// TIA Portal V20 export
// export: Created 2025-12-01T14:57:43.1405238Z, ExportSetting None, DisplayName Totally Integrated Automation Portal, DisplayVersion V20 Update 3, DisplayName TIA Portal Openness, DisplayVersion V20 Update 3, DisplayName TIA Portal Version Control Interface, DisplayVersion V20 Update 3, DisplayName STEP 7 Professional, DisplayVersion V20 Update 3, DisplayName STEP 7 Safety, DisplayVersion V20 Update 2, DisplayName WinCC Basic/Comfort/Advanced, DisplayVersion V20 Update 3, DisplayName WinCC Professional, DisplayVersion V20 Update 3, DisplayName WinCC Unified, DisplayVersion V20 Update 3
DATA_BLOCK "DB1903_ASI_DIAG"   // DB1903
{ S7_Optimized_Access := 'FALSE'; DB_Accessible_From_OPC_UA := 'FALSE' }
// stored: AutoNumber false, DBAccessibleFromOPCUA false
   VAR
      ASI_Gateway_Error : Bool;
      IP_GW { S7_SetPoint := 'True'} : Array[1..16] of "ASI_GW_DATOS";
      ASI3_GW_C1 : Array[1..16] of "ASI3_Diag_GW";
      ASI3_GW_C2 : Array[1..16] of "ASI3_Diag_GW";
      ASI5_GW_Flags { S7_SetPoint := 'True'} : Array[1..16] of "ASI5_Flags";
      ASI5_GW_C1 : Array[1..16] of "ASI5_Diag_GW";
      ASI5_GW_C2 : Array[1..16] of "ASI5_Diag_GW";
   END_VAR
BEGIN
END_DATA_BLOCK
